{attribute addProperty BoxType "IODEVICETYPE_ETHERCATPROT"}
{attribute addProperty Id "SlaveCountAT %I*UINT1620DevStateAT %I*UINT1620Frm0StateAT %I*UINT1620Frm0WcStateAT %I*UINT1620Frm0InputToggleAT %I*UINT1620Frm1StateAT %I*UINT1620Frm1WcStateAT %I*UINT1620Frm1InputToggleAT %I*UINT1620Frm2StateAT %I*UINT1620Frm2WcStateAT %I*UINT1620Frm2InputToggleAT %I*UINT1620Frm3StateAT %I*UINT1620Frm3WcStateAT %I*UINT1620Frm3InputToggleAT %I*UINT1620Frm4StateAT %I*UINT1620Frm4WcStateAT %I*UINT1620Frm4InputToggleAT %I*UINT1620Frm5StateAT %I*UINT1620Frm5WcStateAT %I*UINT1620Frm5InputToggleAT %I*UINT1620Frm6StateAT %I*UINT1620Frm6WcStateAT %I*UINT1620Frm6InputToggleAT %I*UINT1620Frm7StateAT %I*UINT1620Frm7WcStateAT %I*UINT1620Frm7InputToggleAT %I*UINT1620Frm8StateAT %I*UINT1620Frm8WcStateAT %I*UINT1620Frm8InputToggleAT %I*UINT1620Frm9StateAT %I*UINT1620Frm9WcStateAT %I*UINT1620Frm9InputToggleAT %I*UINT1620Frm10StateAT %I*UINT1620Frm10WcStateAT %I*UINT1620Frm10InputToggleAT %I*UINT1620Frm11StateAT %I*UINT1620Frm11WcStateAT %I*UINT1620Frm11InputToggleAT %I*UINT1620Frm12StateAT %I*UINT1620Frm12WcStateAT %I*UINT1620Frm12InputToggleAT %I*UINT1620Frm13StateAT %I*UINT1620Frm13WcStateAT %I*UINT1620Frm13InputToggleAT %I*UINT1620Frm14StateAT %I*UINT1620Frm14WcStateAT %I*UINT1620Frm14InputToggleAT %I*UINT1620Frm15StateAT %I*UINT1620Frm15WcStateAT %I*UINT1620Frm15InputToggleAT %I*UINT1620Frm16StateAT %I*UINT1620Frm16WcStateAT %I*UINT1620Frm16InputToggleAT %I*UINT1620Frm17StateAT %I*UINT1620Frm17WcStateAT %I*UINT1620Frm17InputToggleAT %I*UINT1620Frm18StateAT %I*UINT1620Frm18WcStateAT %I*UINT1620Frm18InputToggleAT %I*UINT1620Frm19StateAT %I*UINT1620Frm19WcStateAT %I*UINT1620Frm19InputToggleAT %I*UINT1620Frm20StateAT %I*UINT1620Frm20WcStateAT %I*UINT1620Frm20InputToggleAT %I*UINT1620Frm21StateAT %I*UINT1620Frm21WcStateAT %I*UINT1620Frm21InputToggleAT %I*UINT1620"}
{attribute addProperty CRC "3272818568"}
{attribute addProperty SizeInBites "1088"}
{attribute addProperty SizeInBytes "136"}
TYPE Inputs_C3133F88 :
STRUCT
	{attribute addProperty Name "SlaveCount"}
	SlaveCount AT %I* : UINT;
	{attribute addProperty Name "DevState"}
	DevState AT %I* : UINT;
	{attribute addProperty Name "Frm0State"}
	Frm0State AT %I* : UINT;
	{attribute addProperty Name "Frm0WcState"}
	Frm0WcState AT %I* : UINT;
	{attribute addProperty Name "Frm0InputToggle"}
	Frm0InputToggle AT %I* : UINT;
	{attribute addProperty Name "Frm1State"}
	Frm1State AT %I* : UINT;
	{attribute addProperty Name "Frm1WcState"}
	Frm1WcState AT %I* : UINT;
	{attribute addProperty Name "Frm1InputToggle"}
	Frm1InputToggle AT %I* : UINT;
	{attribute addProperty Name "Frm2State"}
	Frm2State AT %I* : UINT;
	{attribute addProperty Name "Frm2WcState"}
	Frm2WcState AT %I* : UINT;
	{attribute addProperty Name "Frm2InputToggle"}
	Frm2InputToggle AT %I* : UINT;
	{attribute addProperty Name "Frm3State"}
	Frm3State AT %I* : UINT;
	{attribute addProperty Name "Frm3WcState"}
	Frm3WcState AT %I* : UINT;
	{attribute addProperty Name "Frm3InputToggle"}
	Frm3InputToggle AT %I* : UINT;
	{attribute addProperty Name "Frm4State"}
	Frm4State AT %I* : UINT;
	{attribute addProperty Name "Frm4WcState"}
	Frm4WcState AT %I* : UINT;
	{attribute addProperty Name "Frm4InputToggle"}
	Frm4InputToggle AT %I* : UINT;
	{attribute addProperty Name "Frm5State"}
	Frm5State AT %I* : UINT;
	{attribute addProperty Name "Frm5WcState"}
	Frm5WcState AT %I* : UINT;
	{attribute addProperty Name "Frm5InputToggle"}
	Frm5InputToggle AT %I* : UINT;
	{attribute addProperty Name "Frm6State"}
	Frm6State AT %I* : UINT;
	{attribute addProperty Name "Frm6WcState"}
	Frm6WcState AT %I* : UINT;
	{attribute addProperty Name "Frm6InputToggle"}
	Frm6InputToggle AT %I* : UINT;
	{attribute addProperty Name "Frm7State"}
	Frm7State AT %I* : UINT;
	{attribute addProperty Name "Frm7WcState"}
	Frm7WcState AT %I* : UINT;
	{attribute addProperty Name "Frm7InputToggle"}
	Frm7InputToggle AT %I* : UINT;
	{attribute addProperty Name "Frm8State"}
	Frm8State AT %I* : UINT;
	{attribute addProperty Name "Frm8WcState"}
	Frm8WcState AT %I* : UINT;
	{attribute addProperty Name "Frm8InputToggle"}
	Frm8InputToggle AT %I* : UINT;
	{attribute addProperty Name "Frm9State"}
	Frm9State AT %I* : UINT;
	{attribute addProperty Name "Frm9WcState"}
	Frm9WcState AT %I* : UINT;
	{attribute addProperty Name "Frm9InputToggle"}
	Frm9InputToggle AT %I* : UINT;
	{attribute addProperty Name "Frm10State"}
	Frm10State AT %I* : UINT;
	{attribute addProperty Name "Frm10WcState"}
	Frm10WcState AT %I* : UINT;
	{attribute addProperty Name "Frm10InputToggle"}
	Frm10InputToggle AT %I* : UINT;
	{attribute addProperty Name "Frm11State"}
	Frm11State AT %I* : UINT;
	{attribute addProperty Name "Frm11WcState"}
	Frm11WcState AT %I* : UINT;
	{attribute addProperty Name "Frm11InputToggle"}
	Frm11InputToggle AT %I* : UINT;
	{attribute addProperty Name "Frm12State"}
	Frm12State AT %I* : UINT;
	{attribute addProperty Name "Frm12WcState"}
	Frm12WcState AT %I* : UINT;
	{attribute addProperty Name "Frm12InputToggle"}
	Frm12InputToggle AT %I* : UINT;
	{attribute addProperty Name "Frm13State"}
	Frm13State AT %I* : UINT;
	{attribute addProperty Name "Frm13WcState"}
	Frm13WcState AT %I* : UINT;
	{attribute addProperty Name "Frm13InputToggle"}
	Frm13InputToggle AT %I* : UINT;
	{attribute addProperty Name "Frm14State"}
	Frm14State AT %I* : UINT;
	{attribute addProperty Name "Frm14WcState"}
	Frm14WcState AT %I* : UINT;
	{attribute addProperty Name "Frm14InputToggle"}
	Frm14InputToggle AT %I* : UINT;
	{attribute addProperty Name "Frm15State"}
	Frm15State AT %I* : UINT;
	{attribute addProperty Name "Frm15WcState"}
	Frm15WcState AT %I* : UINT;
	{attribute addProperty Name "Frm15InputToggle"}
	Frm15InputToggle AT %I* : UINT;
	{attribute addProperty Name "Frm16State"}
	Frm16State AT %I* : UINT;
	{attribute addProperty Name "Frm16WcState"}
	Frm16WcState AT %I* : UINT;
	{attribute addProperty Name "Frm16InputToggle"}
	Frm16InputToggle AT %I* : UINT;
	{attribute addProperty Name "Frm17State"}
	Frm17State AT %I* : UINT;
	{attribute addProperty Name "Frm17WcState"}
	Frm17WcState AT %I* : UINT;
	{attribute addProperty Name "Frm17InputToggle"}
	Frm17InputToggle AT %I* : UINT;
	{attribute addProperty Name "Frm18State"}
	Frm18State AT %I* : UINT;
	{attribute addProperty Name "Frm18WcState"}
	Frm18WcState AT %I* : UINT;
	{attribute addProperty Name "Frm18InputToggle"}
	Frm18InputToggle AT %I* : UINT;
	{attribute addProperty Name "Frm19State"}
	Frm19State AT %I* : UINT;
	{attribute addProperty Name "Frm19WcState"}
	Frm19WcState AT %I* : UINT;
	{attribute addProperty Name "Frm19InputToggle"}
	Frm19InputToggle AT %I* : UINT;
	{attribute addProperty Name "Frm20State"}
	Frm20State AT %I* : UINT;
	{attribute addProperty Name "Frm20WcState"}
	Frm20WcState AT %I* : UINT;
	{attribute addProperty Name "Frm20InputToggle"}
	Frm20InputToggle AT %I* : UINT;
	{attribute addProperty Name "Frm21State"}
	Frm21State AT %I* : UINT;
	{attribute addProperty Name "Frm21WcState"}
	Frm21WcState AT %I* : UINT;
	{attribute addProperty Name "Frm21InputToggle"}
	Frm21InputToggle AT %I* : UINT;
END_STRUCT
END_TYPE

(* stored: Version 1.2.0.0, ProductVersion 3.1.4024.9
   DUT Inputs_C3133F88: Id {e1825602-2836-4eef-bfee-2db84725eec0} *)
